FUNCTION_BLOCK Faults5
VAR_INPUT
END_VAR
VAR_OUTPUT
END_VAR
VAR
END_VAR

END_FUNCTION_BLOCK

(* stored: Version 1.1.0.1, ProductVersion 3.1.4024.11
   POU Faults5: Id {15c86bd7-c3d2-4640-85c3-db20ee55a3cc}, SpecialFunc None *)
